FUNCTION_BLOCK PIOC (* Composite Function Block Type *)
  (* Standard: 61499-2 *)
  (* Version 0.0, 12/10/2023, Cheyan, Schneider Electric, template *)
  PACKAGE Main;
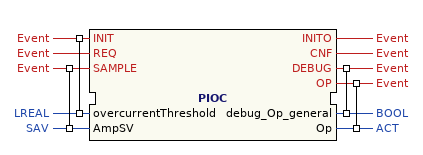
  EVENT_INPUT
    INIT WITH overcurrentThreshold; (* Initialization Request *)
    REQ; (* Normal Execution Request *)
    SAMPLE WITH AmpSV;
  END_EVENT
  EVENT_OUTPUT
    INITO; (* Initialization Confirm *)
    CNF; (* Execution Confirmation *)
    DEBUG WITH debug_Op_general;
    OP WITH Op;
  END_EVENT
  VAR_INPUT
    overcurrentThreshold : LREAL;
    AmpSV : SAV; (* Input event qualifier *)
  END_VAR
  VAR_OUTPUT
    debug_Op_general : BOOL;
    Op : ACT;
  END_VAR
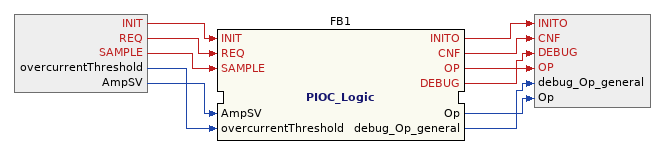
  FBS
    FB1 : PIOC_Logic;
  END_FBS
  EVENT_CONNECTIONS
    INIT TO FB1.INIT;
    REQ TO FB1.REQ;
    FB1.INITO TO INITO;
    FB1.CNF TO CNF;
    FB1.DEBUG TO DEBUG;
    SAMPLE TO FB1.SAMPLE;
    FB1.OP TO OP;
  END_CONNECTIONS
  DATA_CONNECTIONS
    overcurrentThreshold TO FB1.overcurrentThreshold;
    FB1.debug_Op_general TO debug_Op_general;
    AmpSV TO FB1.AmpSV;
    FB1.Op TO Op;
  END_CONNECTIONS
END_FUNCTION_BLOCK
